(* Pump Control *)

FUNCTION_BLOCK FB_Pump
  VAR_INPUT
    Start : BOOL;
    Stop : BOOL;
    Reset : BOOL;
    Fault_In : BOOL;
  END_VAR
  VAR_OUTPUT
    Pump_Run : BOOL;
    Pump_Fault : BOOL;
    Pump_Ready : BOOL;
  END_VAR
  VAR
    sta : BOOL;
  END_VAR

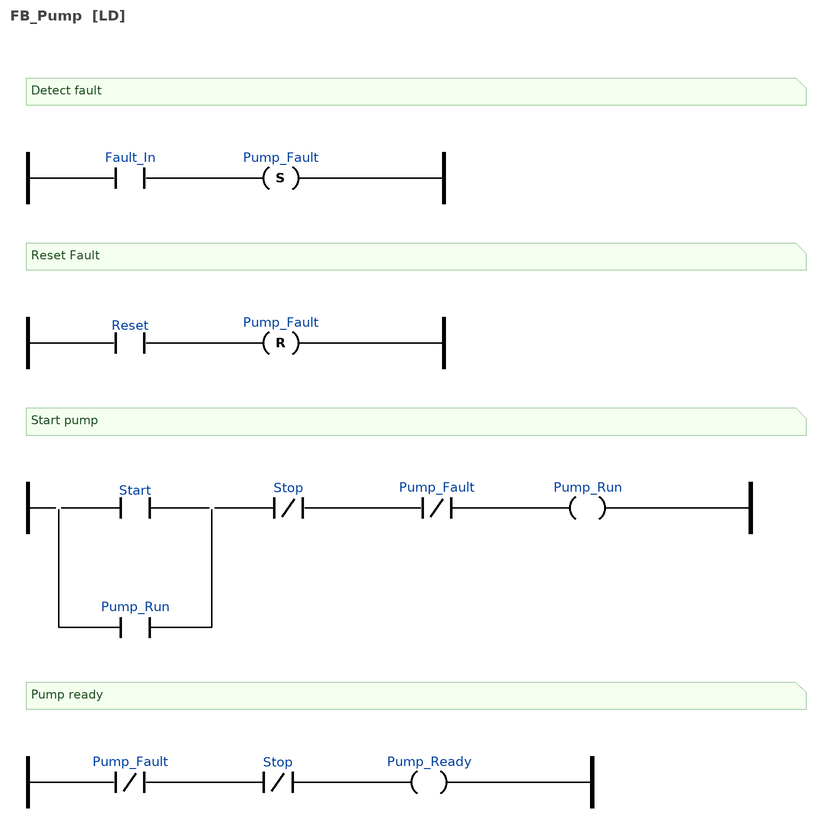
(* LD diagram, written out as Structured Text *)
(* Detect fault *)
IF Fault_In THEN Pump_Fault := TRUE; END_IF;
(* Reset Fault *)
IF Reset THEN Pump_Fault := FALSE; END_IF;
(* Start pump *)
Pump_Run := (Start OR Pump_Run) AND NOT Stop AND NOT Pump_Fault;
(* Pump ready *)
Pump_Ready := NOT Pump_Fault AND NOT Stop;
END_FUNCTION_BLOCK
